(* Logix 5000 project; controller TBIL_All_AOIs_V0_3 vendor 1 type 14 code 176 rev 32.11; software revision 32.00 *)

TASK MainTask (continuous, watchdog 500 ms) : MainProgram
TASK SafetyTask (periodic, rate 20 ms, priority 10, watchdog 20 ms, safety) : SafetyProgram

MODULES
   Local : vendor 1 type 14 code 176 (Compact 0, rev 32.11)
END_MODULES

TYPE Generic_16_Words :
STRUCT
   Data : INT[16];
END_STRUCT
END_TYPE

TYPE Turck_IOLink_Common_Data :
STRUCT
   Read : BOOL;   // For internal use to integrate IOLRead and IOWrite with IOLService
   Write : BOOL;   // For internal use to integrate IOLRead and IOWrite with IOLService
   Reset : BOOL;   // For internal use to integrate IOLRead and IOWrite with IOLService
   Done : BOOL;   // For internal use to integrate IOLRead and IOWrite with IOLService
   Error : BOOL;   // For internal use to integrate IOLRead and IOWrite with IOLService
   Port_in_Use : SINT;   // Each bit is set to show that a port is in use. If it's not in use the port diagnostics will be disabled so IO-Link can still be used but won't throw a red light if no device plugged
   Port : INT;   // For internal use to integrate IOLRead and IOWrite with IOLService
   Index : INT;   // For internal use to integrate IOLRead and IOWrite with IOLService
   SubIndex : INT;   // For internal use to integrate IOLRead and IOWrite with IOLService
   Length : INT;   // For internal use to integrate IOLRead and IOWrite with IOLService
   TicketNum : INT;   // For internal use to integrate IOLRead and IOWrite with IOLService
   Status : INT;   // For internal use to integrate IOLRead and IOWrite with IOLService
   NextTicketNum : INT;   // For internal use to integrate IOLRead and IOWrite with IOLService
   ReceiveData : SINT[255];   // For internal use to integrate IOLRead and IOWrite with IOLService
   SendData : SINT[145];   // For internal use to integrate IOLRead and IOWrite with IOLService
   Vendor_IDs : INT[8];
   Device_IDs : DINT[8];
   WriteData : DINT;
   Process_Input_Data : Generic_16_Words[8];
   Process_Output_Data : Generic_16_Words[8];
END_STRUCT
END_TYPE

ADD_ON_INSTRUCTION IO_Link_Universal_Discrete_Hub   (* revision 1.0 *)
VAR_INPUT
   Port : INT; {required}
END_VAR
VAR_IN_OUT
   Common_Data : Turck_IOLink_Common_Data; {required}
END_VAR
VAR_INPUT
   C0_00_or_7A_Out : BOOL; {visible}
   C0_01_or_7B_Out : BOOL; {visible}
   C1_02_or_5A_Out : BOOL; {visible}
   C1_03_or_5B_Out : BOOL; {visible}
   C2_04_or_3A_Out : BOOL; {visible}
   C2_05_or_3B_Out : BOOL; {visible}
   C3_06_or_1A_Out : BOOL; {visible}
   C3_07_or_1B_Out : BOOL; {visible}
   C4_08_or_8A_Out : BOOL; {visible}
   C4_09_or_8B_Out : BOOL; {visible}
   C5_10_or_6A_Out : BOOL; {visible}
   C5_11_or_6B_Out : BOOL; {visible}
   C6_12_or_4A_Out : BOOL; {visible}
   C6_13_or_4B_Out : BOOL; {visible}
   C7_14_or_2A_Out : BOOL; {visible}
   C7_15_or_2B_Out : BOOL; {visible}
END_VAR
VAR_OUTPUT
   C0_00_or_7A_In : BOOL; {visible}
   C0_01_or_7B_In : BOOL; {visible}
   C1_02_or_5A_In : BOOL; {visible}
   C1_03_or_5B_In : BOOL; {visible}
   C2_04_or_3A_In : BOOL; {visible}
   C2_05_or_3B_In : BOOL; {visible}
   C3_06_or_1A_In : BOOL; {visible}
   C3_07_or_1B_In : BOOL; {visible}
   C4_08_or_8A_In : BOOL; {visible}
   C4_09_or_8B_In : BOOL; {visible}
   C5_10_or_6A_In : BOOL; {visible}
   C5_11_or_6B_In : BOOL; {visible}
   C6_12_or_4A_In : BOOL; {visible}
   C6_13_or_4B_In : BOOL; {visible}
   C7_14_or_2A_In : BOOL; {visible}
   C7_15_or_2B_In : BOOL; {visible}
   TBIL_M1_16DIP : BOOL; {access Read Only}
   TBIL_M1_16DXP : BOOL; {access Read Only}
   TBIL_M1_8DOP : BOOL; {access Read Only}
   TBIL_M1_16DXP_B : BOOL; {access Read Only}
   TBIL_L4_16DXP_AUX : BOOL; {access Read Only}
   TBIL_L5_16DXP_AUX : BOOL;
   TBIL_LL_16DXP_AUX : BOOL; {access Read Only}
   TBIL_S3_8DIP : BOOL; {access Read Only}
   TBIL_S3_8DXP : BOOL; {access Read Only}
   TBIL_S4_8DIP : BOOL; {access Read Only}
   TBIL_S4_8DXP : BOOL; {access Read Only}
   Known_Device_Connected : BOOL; {access Read Only, visible}
   Unknown_Device_or_Missing : BOOL; {access Read Only, visible}
END_VAR
VAR
   Port_Less_One : INT; {access None}
   One : SINT; {access None}
   Port_Bit : SINT; {access None}
   Two : DINT; {access None}
END_VAR

ROUTINE Logic   (* ladder *)
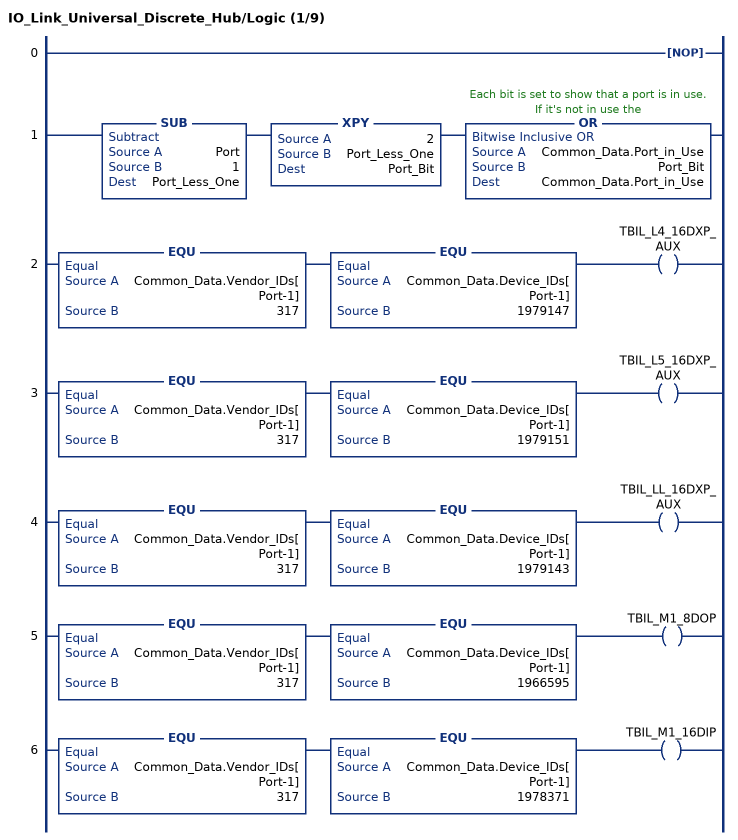
   0: NOP();
   1: SUB(Port,1,Port_Less_One)XPY(2,Port_Less_One,Port_Bit)OR(Common_Data.Port_in_Use,Port_Bit,Common_Data.Port_in_Use);
   2: EQU(Common_Data.Vendor_IDs[Port-1],317)EQU(Common_Data.Device_IDs[Port-1],1979147)OTE(TBIL_L4_16DXP_AUX);
   3: EQU(Common_Data.Vendor_IDs[Port-1],317)EQU(Common_Data.Device_IDs[Port-1],1979151)OTE(TBIL_L5_16DXP_AUX);
   4: EQU(Common_Data.Vendor_IDs[Port-1],317)EQU(Common_Data.Device_IDs[Port-1],1979143)OTE(TBIL_LL_16DXP_AUX);
   5: EQU(Common_Data.Vendor_IDs[Port-1],317)EQU(Common_Data.Device_IDs[Port-1],1966595)OTE(TBIL_M1_8DOP);
   6: EQU(Common_Data.Vendor_IDs[Port-1],317)EQU(Common_Data.Device_IDs[Port-1],1978371)OTE(TBIL_M1_16DIP);
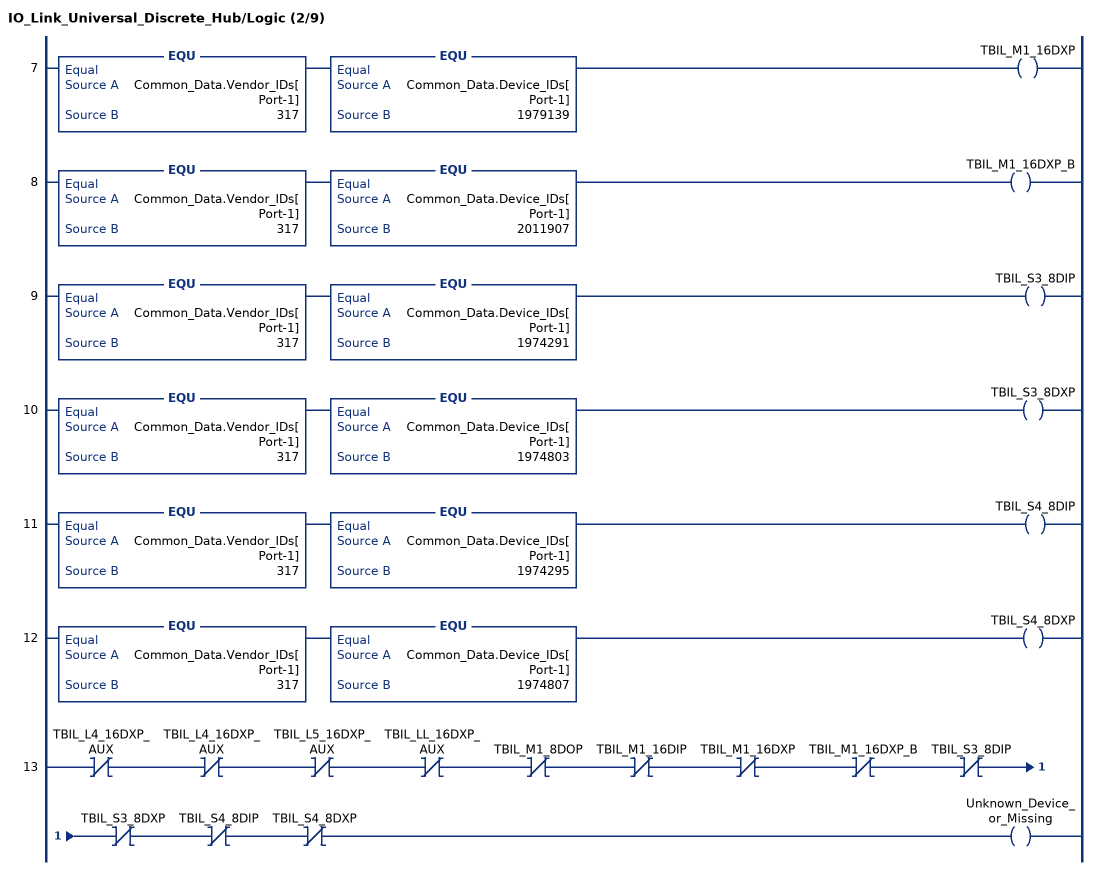
   7: EQU(Common_Data.Vendor_IDs[Port-1],317)EQU(Common_Data.Device_IDs[Port-1],1979139)OTE(TBIL_M1_16DXP);
   8: EQU(Common_Data.Vendor_IDs[Port-1],317)EQU(Common_Data.Device_IDs[Port-1],2011907)OTE(TBIL_M1_16DXP_B);
   9: EQU(Common_Data.Vendor_IDs[Port-1],317)EQU(Common_Data.Device_IDs[Port-1],1974291)OTE(TBIL_S3_8DIP);
   10: EQU(Common_Data.Vendor_IDs[Port-1],317)EQU(Common_Data.Device_IDs[Port-1],1974803)OTE(TBIL_S3_8DXP);
   11: EQU(Common_Data.Vendor_IDs[Port-1],317)EQU(Common_Data.Device_IDs[Port-1],1974295)OTE(TBIL_S4_8DIP);
   12: EQU(Common_Data.Vendor_IDs[Port-1],317)EQU(Common_Data.Device_IDs[Port-1],1974807)OTE(TBIL_S4_8DXP);
   13: XIO(TBIL_L4_16DXP_AUX)XIO(TBIL_L4_16DXP_AUX)XIO(TBIL_L5_16DXP_AUX)XIO(TBIL_LL_16DXP_AUX)XIO(TBIL_M1_8DOP)XIO(TBIL_M1_16DIP)XIO(TBIL_M1_16DXP)XIO(TBIL_M1_16DXP_B)XIO(TBIL_S3_8DIP)XIO(TBIL_S3_8DXP)XIO(TBIL_S4_8DIP)XIO(TBIL_S4_8DXP)OTE(Unknown_Device_or_Missing);
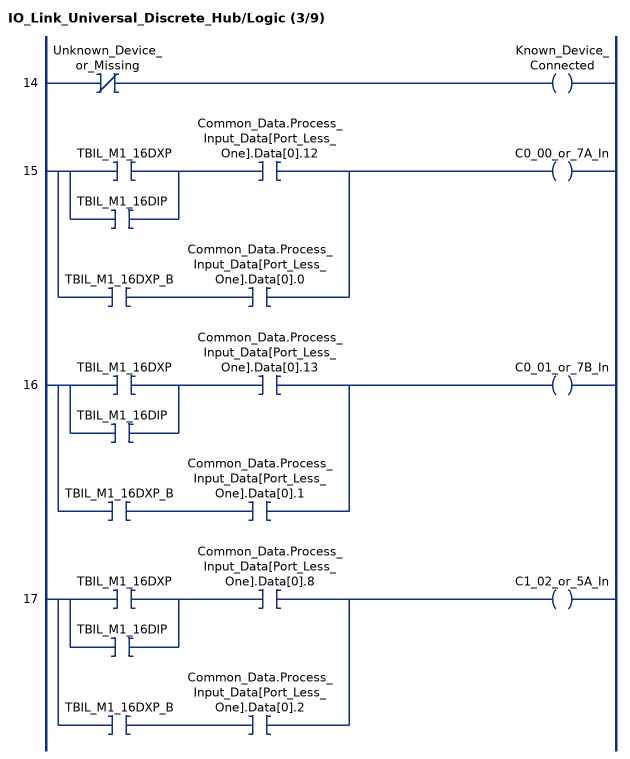
   14: XIO(Unknown_Device_or_Missing)OTE(Known_Device_Connected);
   15: [[XIC(TBIL_M1_16DXP) ,XIC(TBIL_M1_16DIP) ] XIC(Common_Data.Process_Input_Data[Port_Less_One].Data[0].12) ,XIC(TBIL_M1_16DXP_B) XIC(Common_Data.Process_Input_Data[Port_Less_One].Data[0].0) ]OTE(C0_00_or_7A_In);
   16: [[XIC(TBIL_M1_16DXP) ,XIC(TBIL_M1_16DIP) ] XIC(Common_Data.Process_Input_Data[Port_Less_One].Data[0].13) ,XIC(TBIL_M1_16DXP_B) XIC(Common_Data.Process_Input_Data[Port_Less_One].Data[0].1) ]OTE(C0_01_or_7B_In);
   17: [[XIC(TBIL_M1_16DXP) ,XIC(TBIL_M1_16DIP) ] XIC(Common_Data.Process_Input_Data[Port_Less_One].Data[0].8) ,XIC(TBIL_M1_16DXP_B) XIC(Common_Data.Process_Input_Data[Port_Less_One].Data[0].2) ]OTE(C1_02_or_5A_In);
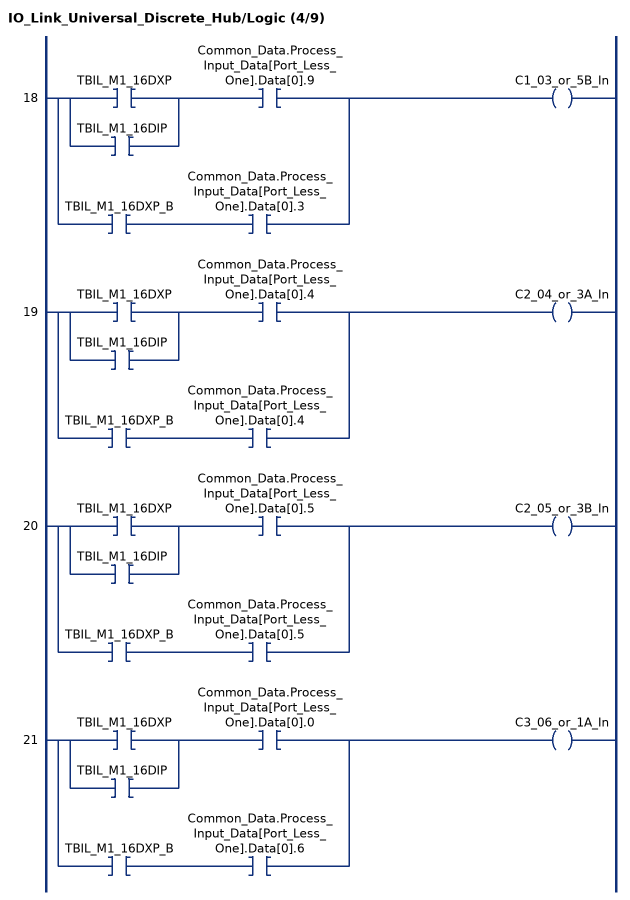
   18: [[XIC(TBIL_M1_16DXP) ,XIC(TBIL_M1_16DIP) ] XIC(Common_Data.Process_Input_Data[Port_Less_One].Data[0].9) ,XIC(TBIL_M1_16DXP_B) XIC(Common_Data.Process_Input_Data[Port_Less_One].Data[0].3) ]OTE(C1_03_or_5B_In);
   19: [[XIC(TBIL_M1_16DXP) ,XIC(TBIL_M1_16DIP) ] XIC(Common_Data.Process_Input_Data[Port_Less_One].Data[0].4) ,XIC(TBIL_M1_16DXP_B) XIC(Common_Data.Process_Input_Data[Port_Less_One].Data[0].4) ]OTE(C2_04_or_3A_In);
   20: [[XIC(TBIL_M1_16DXP) ,XIC(TBIL_M1_16DIP) ] XIC(Common_Data.Process_Input_Data[Port_Less_One].Data[0].5) ,XIC(TBIL_M1_16DXP_B) XIC(Common_Data.Process_Input_Data[Port_Less_One].Data[0].5) ]OTE(C2_05_or_3B_In);
   21: [[XIC(TBIL_M1_16DXP) ,XIC(TBIL_M1_16DIP) ] XIC(Common_Data.Process_Input_Data[Port_Less_One].Data[0].0) ,XIC(TBIL_M1_16DXP_B) XIC(Common_Data.Process_Input_Data[Port_Less_One].Data[0].6) ]OTE(C3_06_or_1A_In);
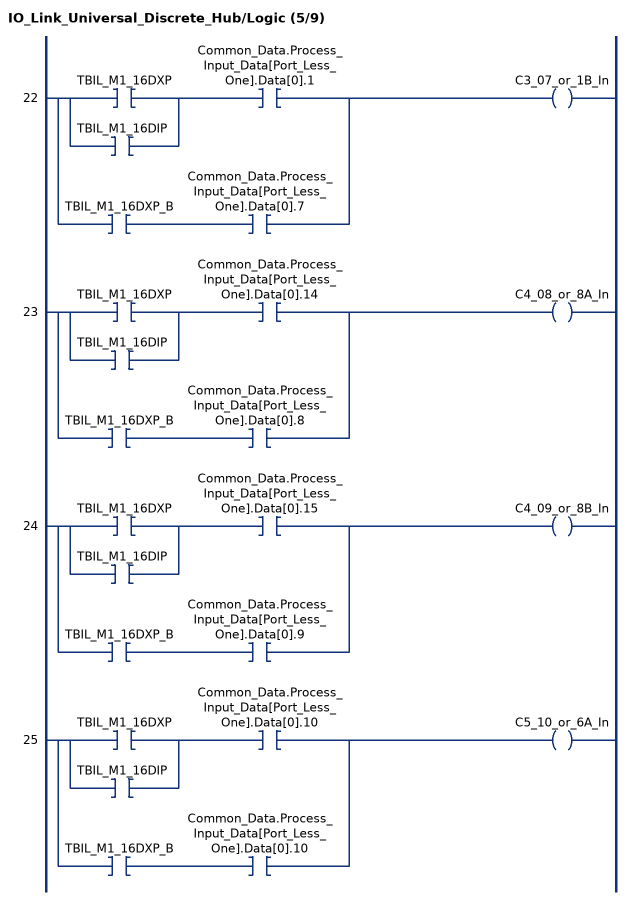
   22: [[XIC(TBIL_M1_16DXP) ,XIC(TBIL_M1_16DIP) ] XIC(Common_Data.Process_Input_Data[Port_Less_One].Data[0].1) ,XIC(TBIL_M1_16DXP_B) XIC(Common_Data.Process_Input_Data[Port_Less_One].Data[0].7) ]OTE(C3_07_or_1B_In);
   23: [[XIC(TBIL_M1_16DXP) ,XIC(TBIL_M1_16DIP) ] XIC(Common_Data.Process_Input_Data[Port_Less_One].Data[0].14) ,XIC(TBIL_M1_16DXP_B) XIC(Common_Data.Process_Input_Data[Port_Less_One].Data[0].8) ]OTE(C4_08_or_8A_In);
   24: [[XIC(TBIL_M1_16DXP) ,XIC(TBIL_M1_16DIP) ] XIC(Common_Data.Process_Input_Data[Port_Less_One].Data[0].15) ,XIC(TBIL_M1_16DXP_B) XIC(Common_Data.Process_Input_Data[Port_Less_One].Data[0].9) ]OTE(C4_09_or_8B_In);
   25: [[XIC(TBIL_M1_16DXP) ,XIC(TBIL_M1_16DIP) ] XIC(Common_Data.Process_Input_Data[Port_Less_One].Data[0].10) ,XIC(TBIL_M1_16DXP_B) XIC(Common_Data.Process_Input_Data[Port_Less_One].Data[0].10) ]OTE(C5_10_or_6A_In);
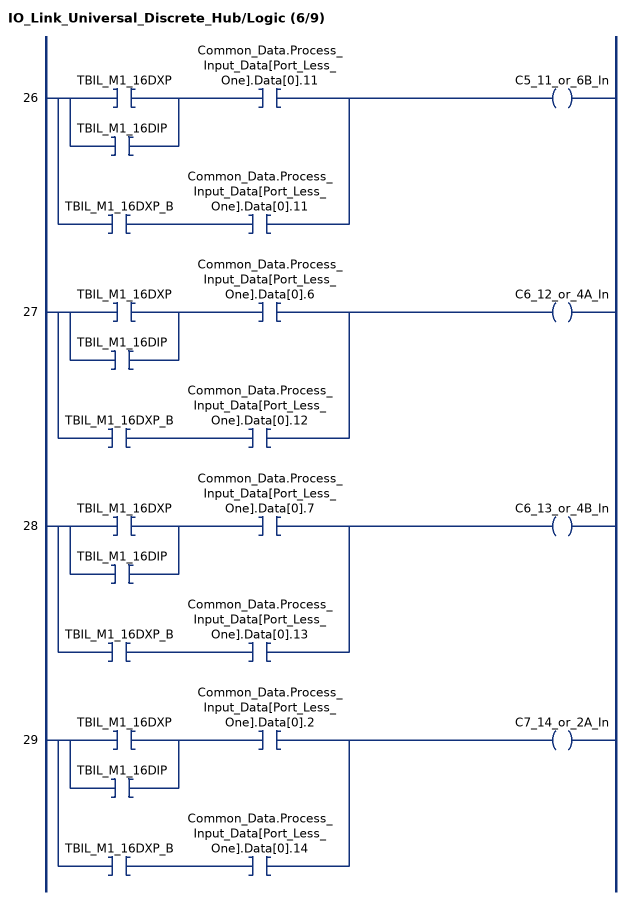
   26: [[XIC(TBIL_M1_16DXP) ,XIC(TBIL_M1_16DIP) ] XIC(Common_Data.Process_Input_Data[Port_Less_One].Data[0].11) ,XIC(TBIL_M1_16DXP_B) XIC(Common_Data.Process_Input_Data[Port_Less_One].Data[0].11) ]OTE(C5_11_or_6B_In);
   27: [[XIC(TBIL_M1_16DXP) ,XIC(TBIL_M1_16DIP) ] XIC(Common_Data.Process_Input_Data[Port_Less_One].Data[0].6) ,XIC(TBIL_M1_16DXP_B) XIC(Common_Data.Process_Input_Data[Port_Less_One].Data[0].12) ]OTE(C6_12_or_4A_In);
   28: [[XIC(TBIL_M1_16DXP) ,XIC(TBIL_M1_16DIP) ] XIC(Common_Data.Process_Input_Data[Port_Less_One].Data[0].7) ,XIC(TBIL_M1_16DXP_B) XIC(Common_Data.Process_Input_Data[Port_Less_One].Data[0].13) ]OTE(C6_13_or_4B_In);
   29: [[XIC(TBIL_M1_16DXP) ,XIC(TBIL_M1_16DIP) ] XIC(Common_Data.Process_Input_Data[Port_Less_One].Data[0].2) ,XIC(TBIL_M1_16DXP_B) XIC(Common_Data.Process_Input_Data[Port_Less_One].Data[0].14) ]OTE(C7_14_or_2A_In);
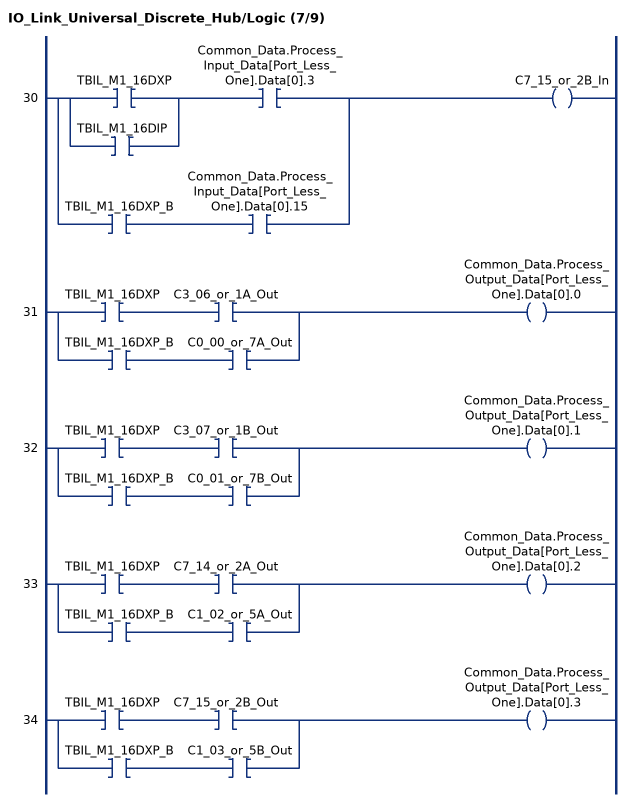
   30: [[XIC(TBIL_M1_16DXP) ,XIC(TBIL_M1_16DIP) ] XIC(Common_Data.Process_Input_Data[Port_Less_One].Data[0].3) ,XIC(TBIL_M1_16DXP_B) XIC(Common_Data.Process_Input_Data[Port_Less_One].Data[0].15) ]OTE(C7_15_or_2B_In);
   31: [XIC(TBIL_M1_16DXP) XIC(C3_06_or_1A_Out) ,XIC(TBIL_M1_16DXP_B) XIC(C0_00_or_7A_Out) ]OTE(Common_Data.Process_Output_Data[Port_Less_One].Data[0].0);
   32: [XIC(TBIL_M1_16DXP) XIC(C3_07_or_1B_Out) ,XIC(TBIL_M1_16DXP_B) XIC(C0_01_or_7B_Out) ]OTE(Common_Data.Process_Output_Data[Port_Less_One].Data[0].1);
   33: [XIC(TBIL_M1_16DXP) XIC(C7_14_or_2A_Out) ,XIC(TBIL_M1_16DXP_B) XIC(C1_02_or_5A_Out) ]OTE(Common_Data.Process_Output_Data[Port_Less_One].Data[0].2);
   34: [XIC(TBIL_M1_16DXP) XIC(C7_15_or_2B_Out) ,XIC(TBIL_M1_16DXP_B) XIC(C1_03_or_5B_Out) ]OTE(Common_Data.Process_Output_Data[Port_Less_One].Data[0].3);
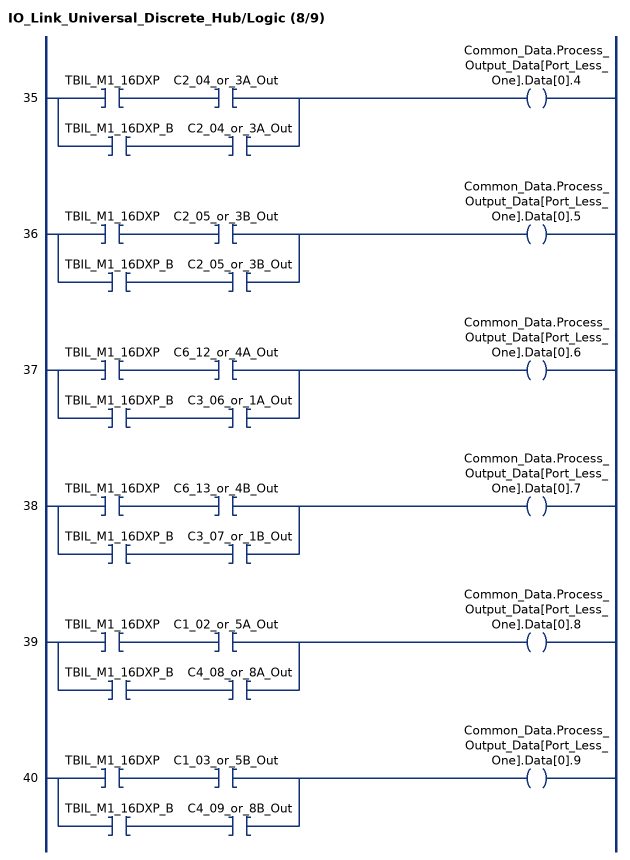
   35: [XIC(TBIL_M1_16DXP) XIC(C2_04_or_3A_Out) ,XIC(TBIL_M1_16DXP_B) XIC(C2_04_or_3A_Out) ]OTE(Common_Data.Process_Output_Data[Port_Less_One].Data[0].4);
   36: [XIC(TBIL_M1_16DXP) XIC(C2_05_or_3B_Out) ,XIC(TBIL_M1_16DXP_B) XIC(C2_05_or_3B_Out) ]OTE(Common_Data.Process_Output_Data[Port_Less_One].Data[0].5);
   37: [XIC(TBIL_M1_16DXP) XIC(C6_12_or_4A_Out) ,XIC(TBIL_M1_16DXP_B) XIC(C3_06_or_1A_Out) ]OTE(Common_Data.Process_Output_Data[Port_Less_One].Data[0].6);
   38: [XIC(TBIL_M1_16DXP) XIC(C6_13_or_4B_Out) ,XIC(TBIL_M1_16DXP_B) XIC(C3_07_or_1B_Out) ]OTE(Common_Data.Process_Output_Data[Port_Less_One].Data[0].7);
   39: [XIC(TBIL_M1_16DXP) XIC(C1_02_or_5A_Out) ,XIC(TBIL_M1_16DXP_B) XIC(C4_08_or_8A_Out) ]OTE(Common_Data.Process_Output_Data[Port_Less_One].Data[0].8);
   40: [XIC(TBIL_M1_16DXP) XIC(C1_03_or_5B_Out) ,XIC(TBIL_M1_16DXP_B) XIC(C4_09_or_8B_Out) ]OTE(Common_Data.Process_Output_Data[Port_Less_One].Data[0].9);
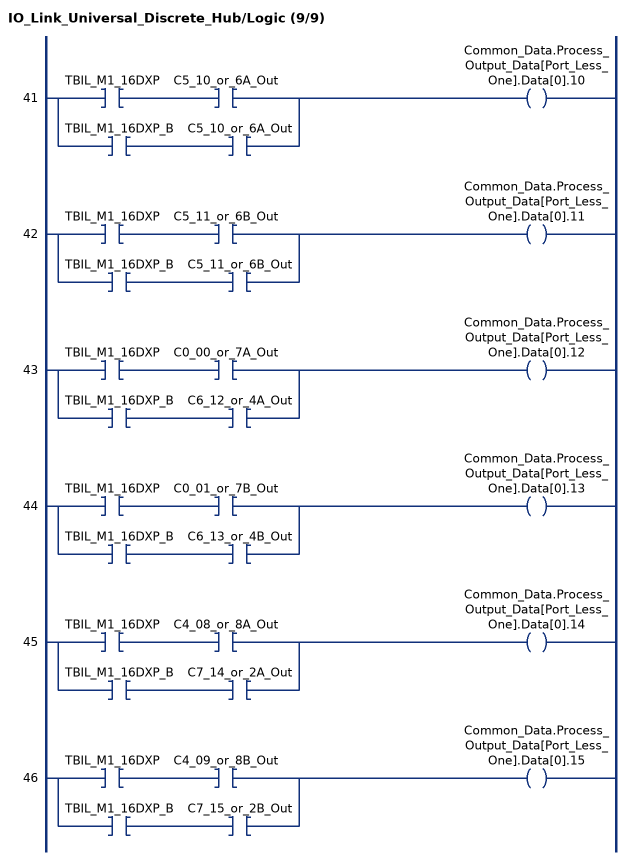
   41: [XIC(TBIL_M1_16DXP) XIC(C5_10_or_6A_Out) ,XIC(TBIL_M1_16DXP_B) XIC(C5_10_or_6A_Out) ]OTE(Common_Data.Process_Output_Data[Port_Less_One].Data[0].10);
   42: [XIC(TBIL_M1_16DXP) XIC(C5_11_or_6B_Out) ,XIC(TBIL_M1_16DXP_B) XIC(C5_11_or_6B_Out) ]OTE(Common_Data.Process_Output_Data[Port_Less_One].Data[0].11);
   43: [XIC(TBIL_M1_16DXP) XIC(C0_00_or_7A_Out) ,XIC(TBIL_M1_16DXP_B) XIC(C6_12_or_4A_Out) ]OTE(Common_Data.Process_Output_Data[Port_Less_One].Data[0].12);
   44: [XIC(TBIL_M1_16DXP) XIC(C0_01_or_7B_Out) ,XIC(TBIL_M1_16DXP_B) XIC(C6_13_or_4B_Out) ]OTE(Common_Data.Process_Output_Data[Port_Less_One].Data[0].13);
   45: [XIC(TBIL_M1_16DXP) XIC(C4_08_or_8A_Out) ,XIC(TBIL_M1_16DXP_B) XIC(C7_14_or_2A_Out) ]OTE(Common_Data.Process_Output_Data[Port_Less_One].Data[0].14);
   46: [XIC(TBIL_M1_16DXP) XIC(C4_09_or_8B_Out) ,XIC(TBIL_M1_16DXP_B) XIC(C7_15_or_2B_Out) ]OTE(Common_Data.Process_Output_Data[Port_Less_One].Data[0].15);
END_ROUTINE
END_ADD_ON_INSTRUCTION

ADD_ON_INSTRUCTION TBEN_Lx_8IOL_AOI   (* revision 0.1 Unreleased, ExecutePrescan *)
// Create an AOI specific to TBEN-Lx-8IOL devices
// Revision note:
// V0_1 Initial Approach
// V0_2 Cleaning Up
// Help:
// IOL_Service - used with Turck BL20, BL67, BLC and TBEN IOLink masters to process requests from IOL_ReadString, IOL_WriteString, IOL_ReadData and IOL_WriteData AOI's.
// Status	Description
// 0	Operation completed successfully
// 	Status = 100 - 102, Ethernet IP MSG instruction errors - check communication parameters
// 100	IOL_SendMSG completed with error, check communication parameters
// 101	IOL_RecevieMSG completed with error, check communication parameters
// 110	IOL_Service Retry Limit exceeded
// 111	Slot specified not an IOLink master
// 	Status = 1000 to 1255, no response from device, connection error
// 1016	Device not connected or Port not configured as IOLink port
// 	Status = 2000 to 2255,  device response indicates error
// 2000	Device error, no details
// 2017	Device error, Index not available
// 2018	Device error, Subindex not available
// 2032	Device error, Service temporarily not available
// 2033	Device error, Service temporarily not available - local control
// 2034	Device error, Service temporarily not available - device control
// 2035	Device error, Index not writeable
// 2048	Device error, Parameter value out of range
// 2049	Device error, Parameter value above limit
// 2050	Device error, Parameter value below limit
// 2051	Device error, Parameter value length overrun (check IOLWrite precision/string length)
// 2052	Device error, Parameter value length underrun (check IOLWrite precision/string length)
// 2053	Device error, Function not available
// 2054	Device error, Function temporarily not available
// 2064	Device error, Parameter set invalid
// 2065	Device error, Inconsistent parameter set
// 2130	Device error, Application not ready
// 	Status = 3000 to 3255,   device response indicates vendor specific error
// 3000	Vendor specific error, no details
// 3001	Vendor specific error, vendor specific error number
// 3255	Vendor specific error, vendor specific error number
// 	Status = 7000 to 7255,  IOL-M Error Codes
// 7000	Unexpected write request instead of read request
// 7001	Decode error
// 7002	Port occupied by another task
// 	Status = 8000 to 8255,  IOL-M Error Codes
// 8000	Timeout when IOL-Ds or IOL-M ports are busy
// 8001	IOL Index out of range
// 8002	Port address greater than maximum
// 8003	Port function not supported
VAR_IN_OUT
   Common_Data : Turck_IOLink_Common_Data; {required}
        .SendData[1]   // For internal use to integrate IOLRead and IOLWrite with IOLService
   IOL_Read_MSG : MESSAGE; {required}
   IOL_Write_MSG : MESSAGE; {required}
   TBEN_I_DATA : INT[173]; {required}   // Input Data from IO Block
   TBEN_O_DATA : INT[131]; {required}   // Output Data to IO Block
   TBEN_C_DATA : SINT[160]; {required}
END_VAR
VAR_OUTPUT
   DXP1_OUT : BOOL; {visible}
   DXP3_OUT : BOOL; {visible}
   DXP5_OUT : BOOL; {visible}
   DXP7_OUT : BOOL; {visible}
   IOLDevice_PORT1 : BOOL; {visible}
   IOLDevice_PORT2 : BOOL; {visible}
   IOLDevice_PORT3 : BOOL; {visible}
   IOLDevice_PORT4 : BOOL; {visible}
   IOLDevice_PORT5 : BOOL; {visible}
   IOLDevice_PORT6 : BOOL; {visible}
   IOLDevice_PORT7 : BOOL; {visible}
   IOLDevice_PORT8 : BOOL; {visible}
END_VAR
VAR_INPUT
   IOL0_DI : BOOL; {visible}
   DXP1_IN : BOOL; {visible}
   IOL2_DI : BOOL; {visible}
   DXP3_IN : BOOL; {visible}
   IOL4_DI : BOOL; {visible}
   DXP5_IN : BOOL; {visible}
   IOL6_DI : BOOL; {visible}
   DXP7_IN : BOOL; {visible}
   IOL8_DI : BOOL; {visible}
   IOL10_DI : BOOL; {visible}
   IOL12_DI : BOOL; {visible}
   IOL14_DI : BOOL; {visible}
   PORT1_Mode_IOL_or_DI : BOOL;   // 0: IO-LINK without validation 1: Port is set to DI (Power Cycle or Module Inhibit cycle require)
   PORT2_Mode_IOL_or_DI : BOOL;   // 0: IO-LINK without validation 1: Port is set to DI (Power Cycle or Module Inhibit cycle require)
   PORT3_Mode_IOL_or_DI : BOOL;   // 0: IO-LINK without validation 1: Port is set to DI (Power Cycle or Module Inhibit cycle require)
   PORT4_Mode_IOL_or_DI : BOOL;   // 0: IO-LINK without validation 1: Port is set to DI (Power Cycle or Module Inhibit cycle require)
   PORT5_Mode_IOL_or_DI : BOOL;   // 0: IO-LINK without validation 1: Port is set to DI (Power Cycle or Module Inhibit cycle require)
   PORT6_Mode_IOL_or_DI : BOOL;   // 0: IO-LINK without validation 1: Port is set to DI (Power Cycle or Module Inhibit cycle require)
   PORT7_Mode_IOL_or_DI : BOOL;   // 0: IO-LINK without validation 1: Port is set to DI (Power Cycle or Module Inhibit cycle require)
   PORT8_Mode_IOL_or_DI : BOOL;   // 0: IO-LINK without validation 1: Port is set to DI (Power Cycle or Module Inhibit cycle require)
   DisableOutput_DXP1 : BOOL;
   DisableOutput_DXP3 : BOOL;
   DisableOutput_DXP5 : BOOL;
   DisableOutput_DXP7 : BOOL;
END_VAR
VAR_OUTPUT
   Device_Restart_Required : BOOL; {visible}
END_VAR
VAR_INPUT
   DeviceStatus : DINT;
END_VAR
VAR
   IOLReadActive : BOOL;
   IOLWriteActive : BOOL;
   RetryCount : DINT;
   IOL_Error_Count : DINT; {access None}
   IOLReset_ONS : BOOL; {access None}
   ER1 : BOOL; {access None}
   ER2 : BOOL; {access None}
   tempReceiveData : SINT[255]; {access None}
   Generate_Status : BOOL; {access None}
   ABS_RD_0 : INT; {access None}
   ABS_RD_1 : INT; {access None}
   ABS_RD_2 : INT; {access None}
   ABS_RD_3 : INT; {access None}
   tempSendData : SINT[145]; {access None}
   IOL_READ_Request : BOOL; {access None}
   IOL_WRITE_Request : BOOL; {access None}
   StartupDone : BOOL; {access None}
   Done : BOOL; {access None}
   Error : BOOL; {access None}
   Active : BOOL; {access None}
   Pending : BOOL; {access None}
   Pending_or_Active : BOOL; {access None}
   StartupCount : SINT; {access None}
   DoneCount : SINT; {access None}
   MyTicketNum : INT; {access None}
   Update_Data : BOOL; {access None}
   Read_ONS : BOOL; {access None}
   ReadRequest : BOOL; {access None}
   Prev_Input_Data_Valids : INT; {access None}
   Status : DINT; {access None}
   ErrorCount : DINT; {access None}
   PIDV_Delay : TIMER := (PRE := 1000); {access None}
   TimeDelay : TIMER := (PRE := 500); {access None}
END_VAR

ROUTINE Logic   (* ladder *)
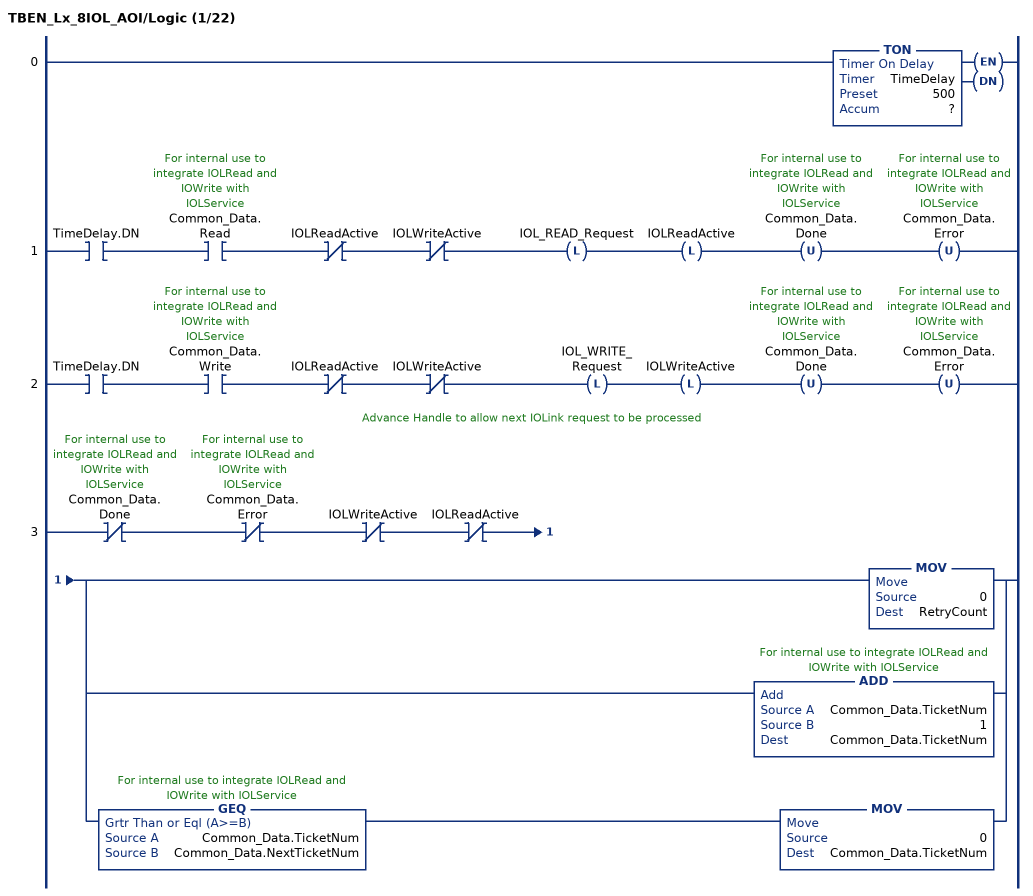
   0: TON(TimeDelay,?,?);
   1: XIC(TimeDelay.DN)XIC(Common_Data.Read)XIO(IOLReadActive)XIO(IOLWriteActive)OTL(IOL_READ_Request)OTL(IOLReadActive)OTU(Common_Data.Done)OTU(Common_Data.Error);
   2: XIC(TimeDelay.DN)XIC(Common_Data.Write)XIO(IOLReadActive)XIO(IOLWriteActive)OTL(IOL_WRITE_Request)OTL(IOLWriteActive)OTU(Common_Data.Done)OTU(Common_Data.Error);
   // Advance Handle to allow next IOLink request to be processed
   3: XIO(Common_Data.Done)XIO(Common_Data.Error)XIO(IOLWriteActive)XIO(IOLReadActive)[MOV(0,RetryCount) ,ADD(Common_Data.TicketNum,1,Common_Data.TicketNum) ,GEQ(Common_Data.TicketNum,Common_Data.NextTicketNum) MOV(0,Common_Data.TicketNum) ];
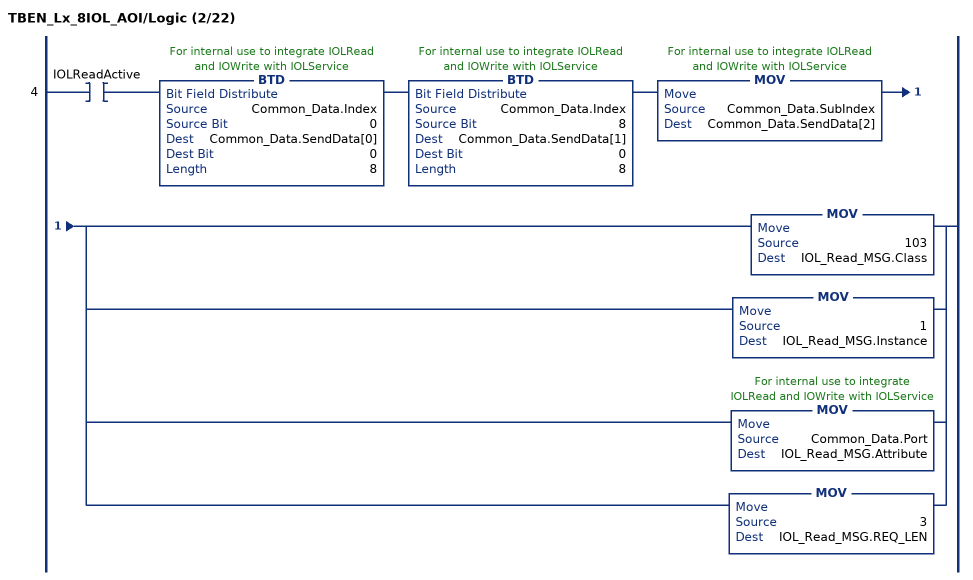
   4: XIC(IOLReadActive)BTD(Common_Data.Index,0,Common_Data.SendData[0],0,8)BTD(Common_Data.Index,8,Common_Data.SendData[1],0,8)MOV(Common_Data.SubIndex,Common_Data.SendData[2])[MOV(103,IOL_Read_MSG.Class) ,MOV(1,IOL_Read_MSG.Instance) ,MOV(Common_Data.Port,IOL_Read_MSG.Attribute) ,MOV(3,IOL_Read_MSG.REQ_LEN) ];
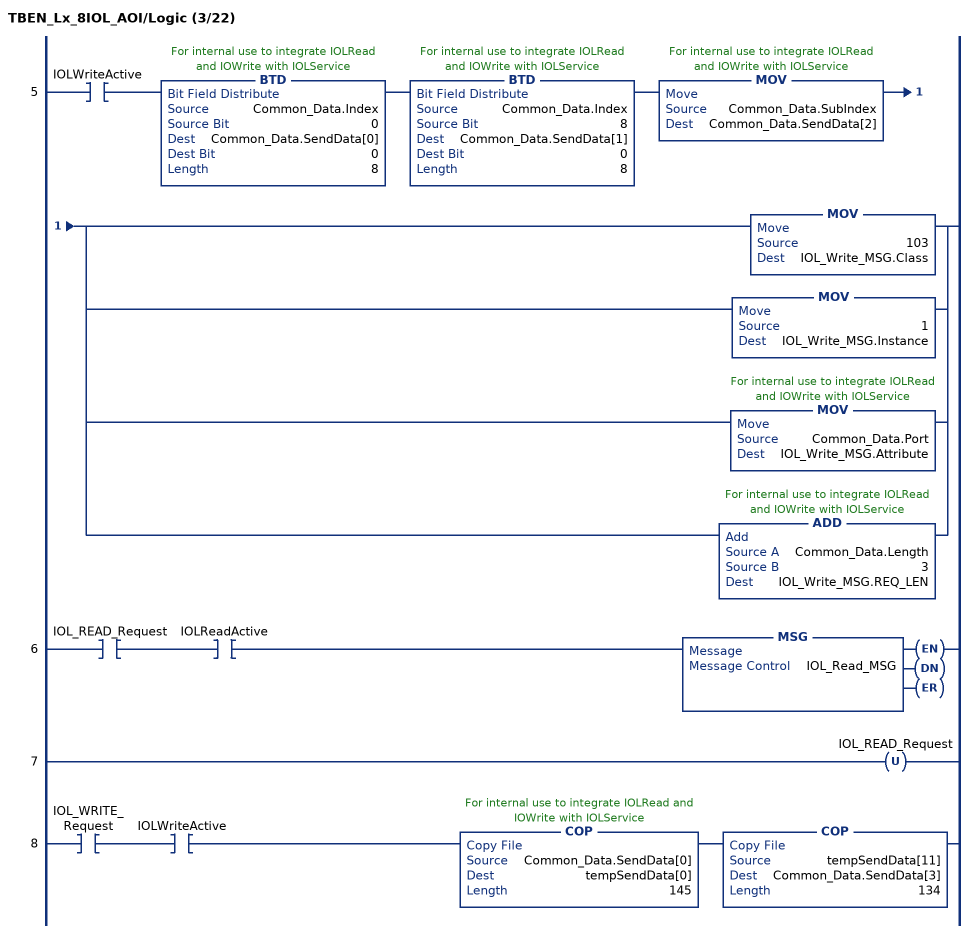
   5: XIC(IOLWriteActive)BTD(Common_Data.Index,0,Common_Data.SendData[0],0,8)BTD(Common_Data.Index,8,Common_Data.SendData[1],0,8)MOV(Common_Data.SubIndex,Common_Data.SendData[2])[MOV(103,IOL_Write_MSG.Class) ,MOV(1,IOL_Write_MSG.Instance) ,MOV(Common_Data.Port,IOL_Write_MSG.Attribute) ,ADD(Common_Data.Length,3,IOL_Write_MSG.REQ_LEN) ];
   6: XIC(IOL_READ_Request)XIC(IOLReadActive)MSG(IOL_Read_MSG);
   7: OTU(IOL_READ_Request);
   8: XIC(IOL_WRITE_Request)XIC(IOLWriteActive)COP(Common_Data.SendData[0],tempSendData[0],145)COP(tempSendData[11],Common_Data.SendData[3],134);
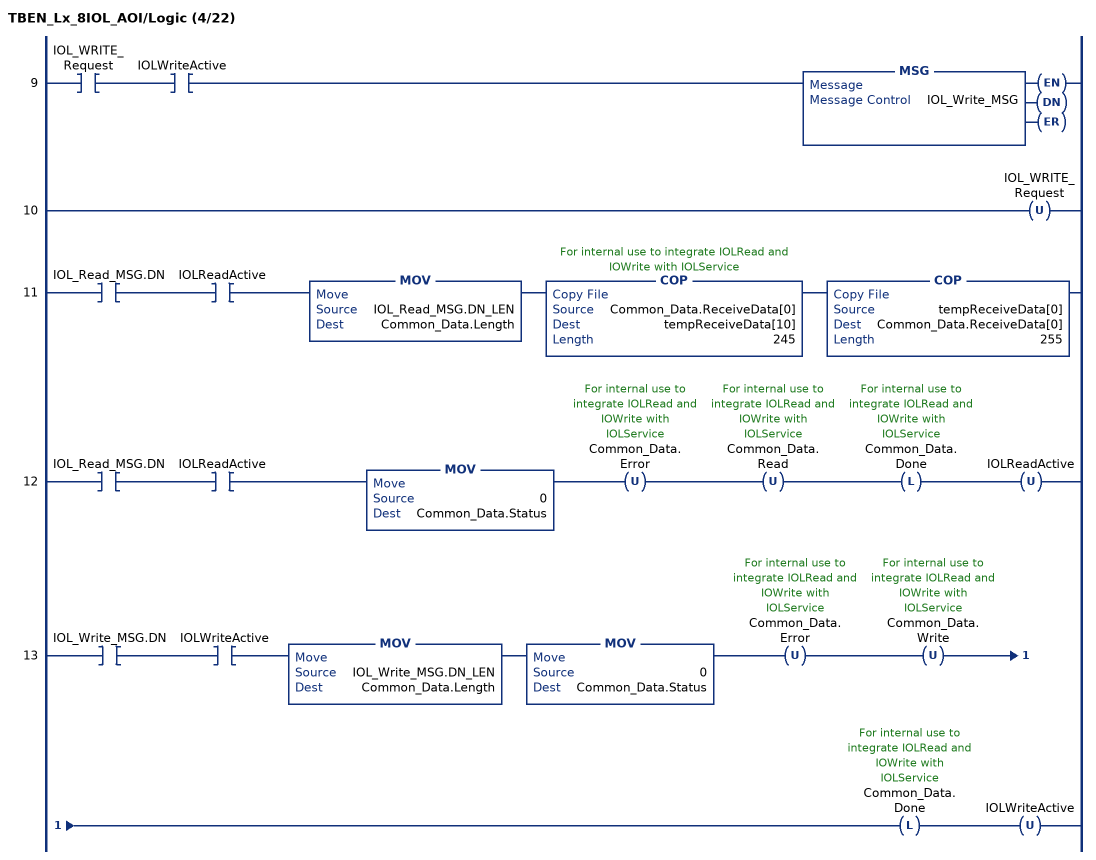
   9: XIC(IOL_WRITE_Request)XIC(IOLWriteActive)MSG(IOL_Write_MSG);
   10: OTU(IOL_WRITE_Request);
   11: XIC(IOL_Read_MSG.DN)XIC(IOLReadActive)MOV(IOL_Read_MSG.DN_LEN,Common_Data.Length)COP(Common_Data.ReceiveData[0],tempReceiveData[10],245)COP(tempReceiveData[0],Common_Data.ReceiveData[0],255);
   12: XIC(IOL_Read_MSG.DN)XIC(IOLReadActive)MOV(0,Common_Data.Status)OTU(Common_Data.Error)OTU(Common_Data.Read)OTL(Common_Data.Done)OTU(IOLReadActive);
   13: XIC(IOL_Write_MSG.DN)XIC(IOLWriteActive)MOV(IOL_Write_MSG.DN_LEN,Common_Data.Length)MOV(0,Common_Data.Status)OTU(Common_Data.Error)OTU(Common_Data.Write)OTL(Common_Data.Done)OTU(IOLWriteActive);
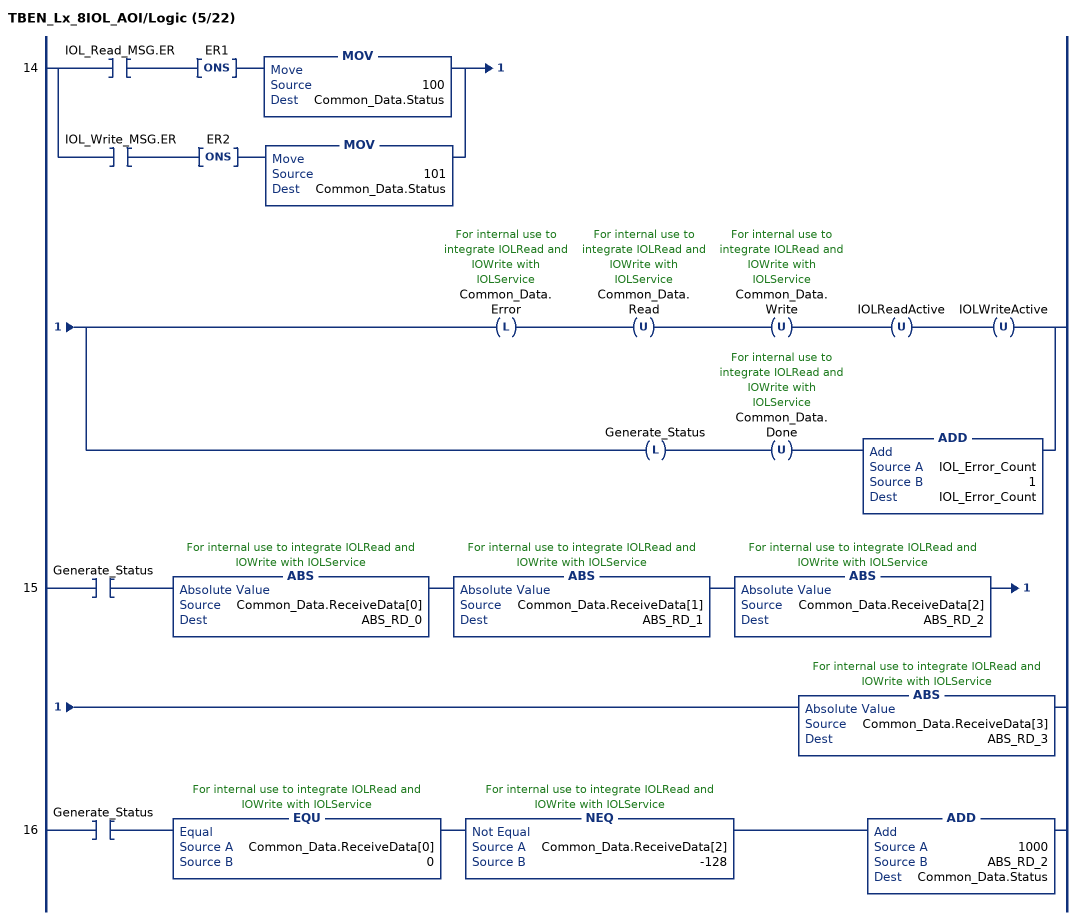
   14: [XIC(IOL_Read_MSG.ER) ONS(ER1) MOV(100,Common_Data.Status) ,XIC(IOL_Write_MSG.ER) ONS(ER2) MOV(101,Common_Data.Status) ][OTL(Common_Data.Error) OTU(Common_Data.Read) OTU(Common_Data.Write) OTU(IOLReadActive) OTU(IOLWriteActive) ,OTL(Generate_Status) OTU(Common_Data.Done) ADD(IOL_Error_Count,1,IOL_Error_Count) ];
   15: XIC(Generate_Status)ABS(Common_Data.ReceiveData[0],ABS_RD_0)ABS(Common_Data.ReceiveData[1],ABS_RD_1)ABS(Common_Data.ReceiveData[2],ABS_RD_2)ABS(Common_Data.ReceiveData[3],ABS_RD_3);
   16: XIC(Generate_Status)EQU(Common_Data.ReceiveData[0],0)NEQ(Common_Data.ReceiveData[2],-128)ADD(1000,ABS_RD_2,Common_Data.Status);
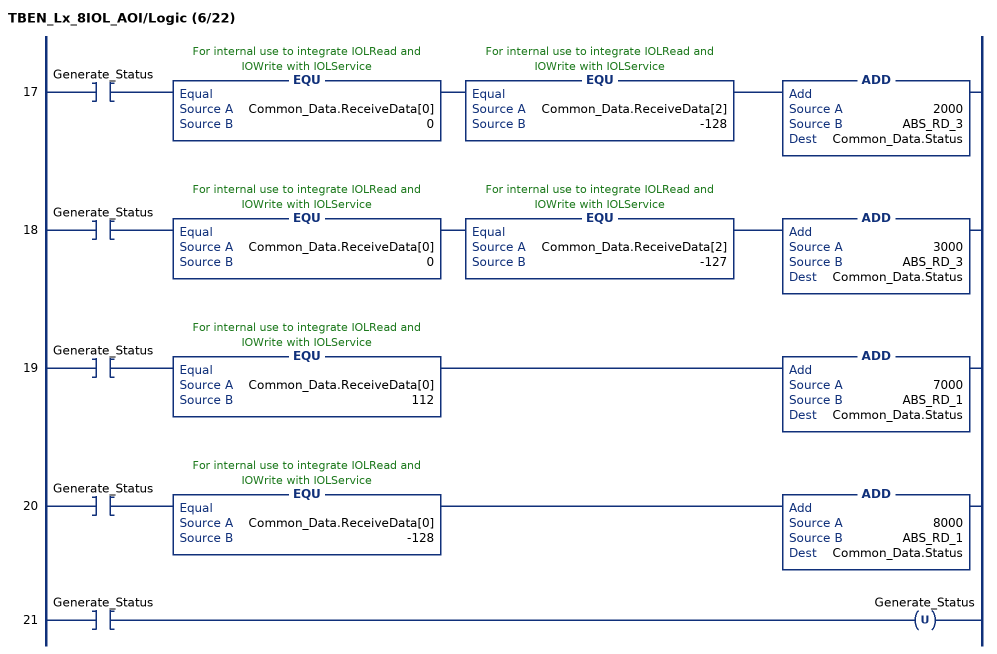
   17: XIC(Generate_Status)EQU(Common_Data.ReceiveData[0],0)EQU(Common_Data.ReceiveData[2],-128)ADD(2000,ABS_RD_3,Common_Data.Status);
   18: XIC(Generate_Status)EQU(Common_Data.ReceiveData[0],0)EQU(Common_Data.ReceiveData[2],-127)ADD(3000,ABS_RD_3,Common_Data.Status);
   19: XIC(Generate_Status)EQU(Common_Data.ReceiveData[0],112)ADD(7000,ABS_RD_1,Common_Data.Status);
   20: XIC(Generate_Status)EQU(Common_Data.ReceiveData[0],-128)ADD(8000,ABS_RD_1,Common_Data.Status);
   21: XIC(Generate_Status)OTU(Generate_Status);
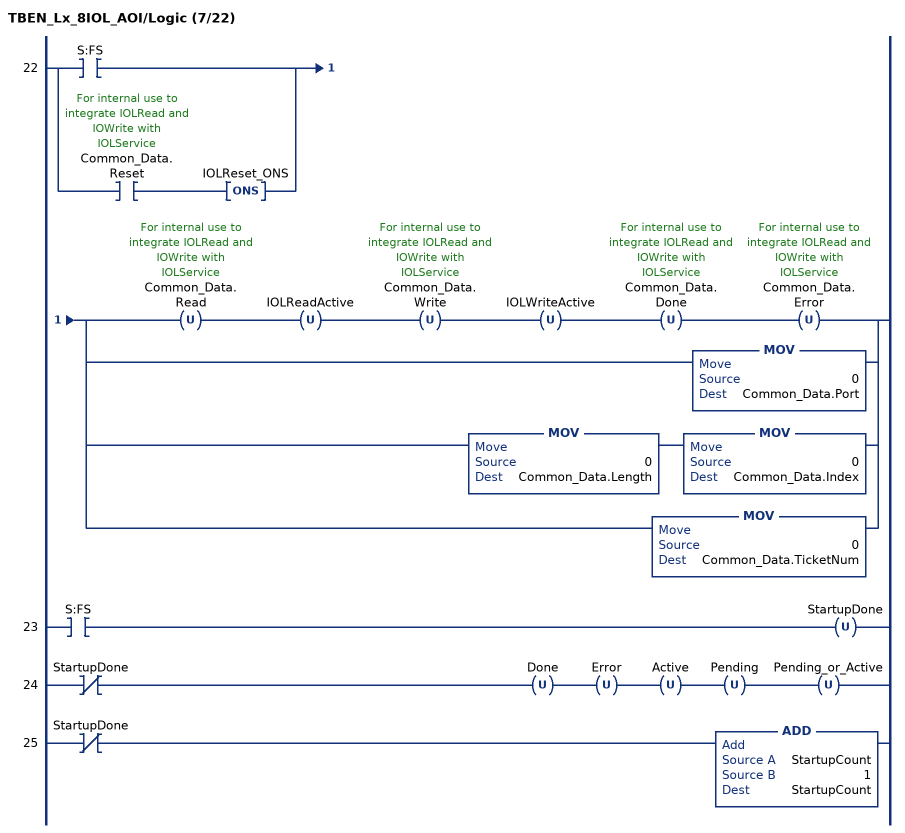
   22: [XIC(S:FS) ,XIC(Common_Data.Reset) ONS(IOLReset_ONS) ][OTU(Common_Data.Read) OTU(IOLReadActive) OTU(Common_Data.Write) OTU(IOLWriteActive) OTU(Common_Data.Done) OTU(Common_Data.Error) ,MOV(0,Common_Data.Port) ,MOV(0,Common_Data.Length) MOV(0,Common_Data.Index) ,MOV(0,Common_Data.TicketNum) ];
   23: XIC(S:FS)OTU(StartupDone);
   24: XIO(StartupDone)OTU(Done)OTU(Error)OTU(Active)OTU(Pending)OTU(Pending_or_Active);
   25: XIO(StartupDone)ADD(StartupCount,1,StartupCount);
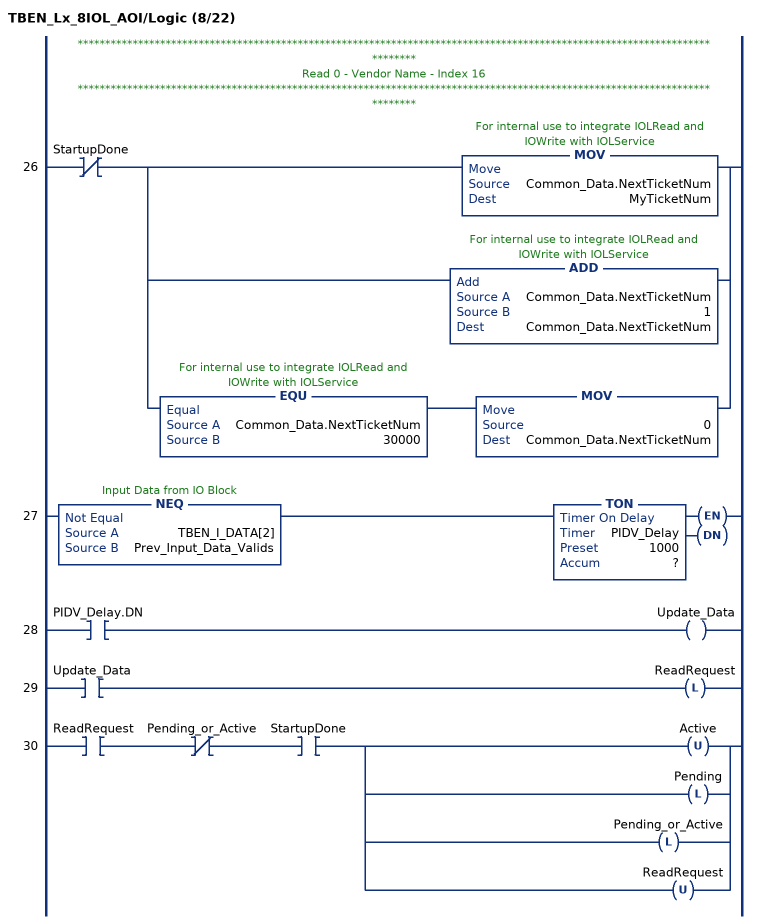
   // ***************************************************************************************************************************
   // Read 0 - Vendor Name - Index 16
   // ***************************************************************************************************************************
   26: XIO(StartupDone)[MOV(Common_Data.NextTicketNum,MyTicketNum) ,ADD(Common_Data.NextTicketNum,1,Common_Data.NextTicketNum) ,EQU(Common_Data.NextTicketNum,30000) MOV(0,Common_Data.NextTicketNum) ];
   27: NEQ(TBEN_I_DATA[2],Prev_Input_Data_Valids)TON(PIDV_Delay,?,?);
   28: XIC(PIDV_Delay.DN)OTE(Update_Data);
   29: XIC(Update_Data)OTL(ReadRequest);
   30: XIC(ReadRequest)XIO(Pending_or_Active)XIC(StartupDone)[OTU(Active) ,OTL(Pending) ,OTL(Pending_or_Active) ,OTU(ReadRequest) ];
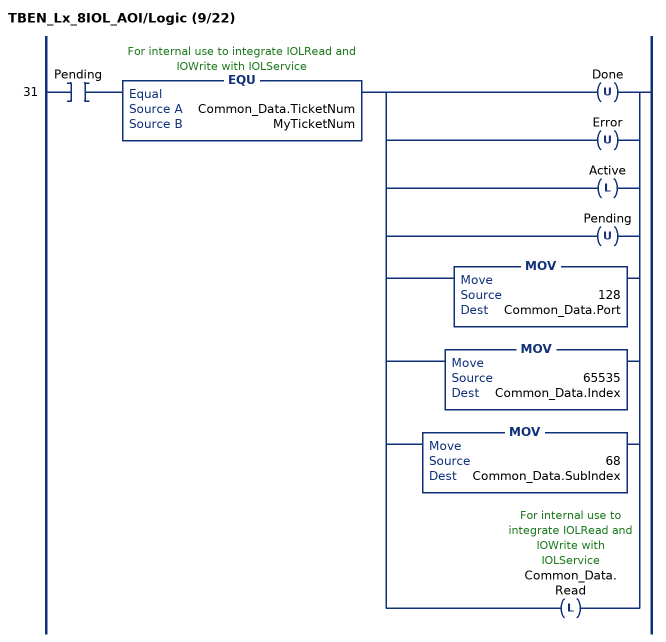
   31: XIC(Pending)EQU(Common_Data.TicketNum,MyTicketNum)[OTU(Done) ,OTU(Error) ,OTL(Active) ,OTU(Pending) ,MOV(128,Common_Data.Port) ,MOV(65535,Common_Data.Index) ,MOV(68,Common_Data.SubIndex) ,OTL(Common_Data.Read) ];
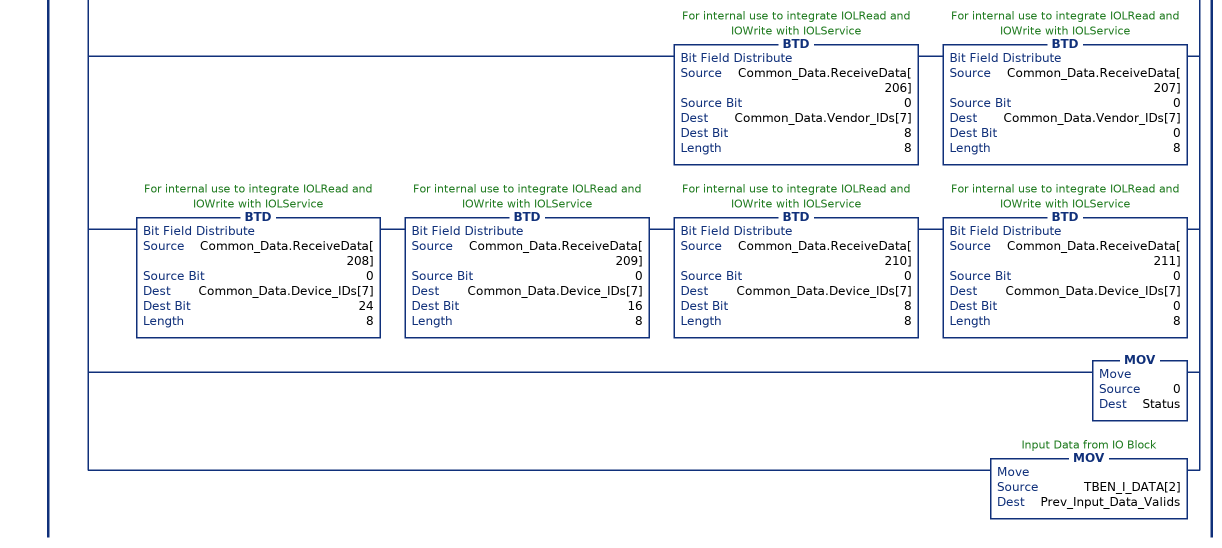
   32: XIC(Active)XIC(Common_Data.Done)[OTL(Done) ,ADD(DoneCount,1,DoneCount) ,OTU(Error) ,OTU(Active) ,OTU(Pending) ,OTU(Pending_or_Active) ,OTU(Common_Data.Done) ,BTD(Common_Data.ReceiveData[10],0,Common_Data.Vendor_IDs[0],8,8) BTD(Common_Data.ReceiveData[11],0,Common_Data.Vendor_IDs[0],0,8) ,BTD(Common_Data.ReceiveData[12],0,Common_Data.Device_IDs[0],24,8) BTD(Common_Data.ReceiveData[13],0,Common_Data.Device_IDs[0],16,8) BTD(Common_Data.ReceiveData[14],0,Common_Data.Device_IDs[0],8,8) BTD(Common_Data.ReceiveData[15],0,Common_Data.Device_IDs[0],0,8) ,BTD(Common_Data.ReceiveData[38],0,Common_Data.Vendor_IDs[1],8,8) BTD(Common_Data.ReceiveData[39],0,Common_Data.Vendor_IDs[1],0,8) ,BTD(Common_Data.ReceiveData[40],0,Common_Data.Device_IDs[1],24,8) BTD(Common_Data.ReceiveData[41],0,Common_Data.Device_IDs[1],16,8) BTD(Common_Data.ReceiveData[42],0,Common_Data.Device_IDs[1],8,8) BTD(Common_Data.ReceiveData[43],0,Common_Data.Device_IDs[1],0,8) ,BTD(Common_Data.ReceiveData[66],0,Common_Data.Vendor_IDs[2],8,8) BTD(Common_Data.ReceiveData[67],0,Common_Data.Vendor_IDs[2],0,8) ,BTD(Common_Data.ReceiveData[68],0,Common_Data.Device_IDs[2],24,8) BTD(Common_Data.ReceiveData[69],0,Common_Data.Device_IDs[2],16,8) BTD(Common_Data.ReceiveData[70],0,Common_Data.Device_IDs[2],8,8) BTD(Common_Data.ReceiveData[71],0,Common_Data.Device_IDs[2],0,8) ,BTD(Common_Data.ReceiveData[94],0,Common_Data.Vendor_IDs[3],8,8) BTD(Common_Data.ReceiveData[95],0,Common_Data.Vendor_IDs[3],0,8) ,BTD(Common_Data.ReceiveData[96],0,Common_Data.Device_IDs[3],24,8) BTD(Common_Data.ReceiveData[97],0,Common_Data.Device_IDs[3],16,8) BTD(Common_Data.ReceiveData[98],0,Common_Data.Device_IDs[3],8,8) BTD(Common_Data.ReceiveData[99],0,Common_Data.Device_IDs[3],0,8) ,BTD(Common_Data.ReceiveData[122],0,Common_Data.Vendor_IDs[4],8,8) BTD(Common_Data.ReceiveData[123],0,Common_Data.Vendor_IDs[4],0,8) ,BTD(Common_Data.ReceiveData[124],0,Common_Data.Device_IDs[4],24,8) BTD(Common_Data.ReceiveData[125],0,Common_Data.Device_IDs[4],16,8) BTD(Common_Data.ReceiveData[126],0,Common_Data.Device_IDs[4],8,8) BTD(Common_Data.ReceiveData[127],0,Common_Data.Device_IDs[4],0,8) ,BTD(Common_Data.ReceiveData[150],0,Common_Data.Vendor_IDs[5],8,8) BTD(Common_Data.ReceiveData[151],0,Common_Data.Vendor_IDs[5],0,8) ,BTD(Common_Data.ReceiveData[152],0,Common_Data.Device_IDs[5],24,8) BTD(Common_Data.ReceiveData[153],0,Common_Data.Device_IDs[5],16,8) BTD(Common_Data.ReceiveData[154],0,Common_Data.Device_IDs[5],8,8) BTD(Common_Data.ReceiveData[155],0,Common_Data.Device_IDs[5],0,8) ,BTD(Common_Data.ReceiveData[178],0,Common_Data.Vendor_IDs[6],8,8) BTD(Common_Data.ReceiveData[179],0,Common_Data.Vendor_IDs[6],0,8) ,BTD(Common_Data.ReceiveData[180],0,Common_Data.Device_IDs[6],24,8) BTD(Common_Data.ReceiveData[181],0,Common_Data.Device_IDs[6],16,8) BTD(Common_Data.ReceiveData[182],0,Common_Data.Device_IDs[6],8,8) BTD(Common_Data.ReceiveData[183],0,Common_Data.Device_IDs[6],0,8) ,BTD(Common_Data.ReceiveData[206],0,Common_Data.Vendor_IDs[7],8,8) BTD(Common_Data.ReceiveData[207],0,Common_Data.Vendor_IDs[7],0,8) ,BTD(Common_Data.ReceiveData[208],0,Common_Data.Device_IDs[7],24,8) BTD(Common_Data.ReceiveData[209],0,Common_Data.Device_IDs[7],16,8) BTD(Common_Data.ReceiveData[210],0,Common_Data.Device_IDs[7],8,8) BTD(Common_Data.ReceiveData[211],0,Common_Data.Device_IDs[7],0,8) ,MOV(0,Status) ,MOV(TBEN_I_DATA[2],Prev_Input_Data_Valids) ];
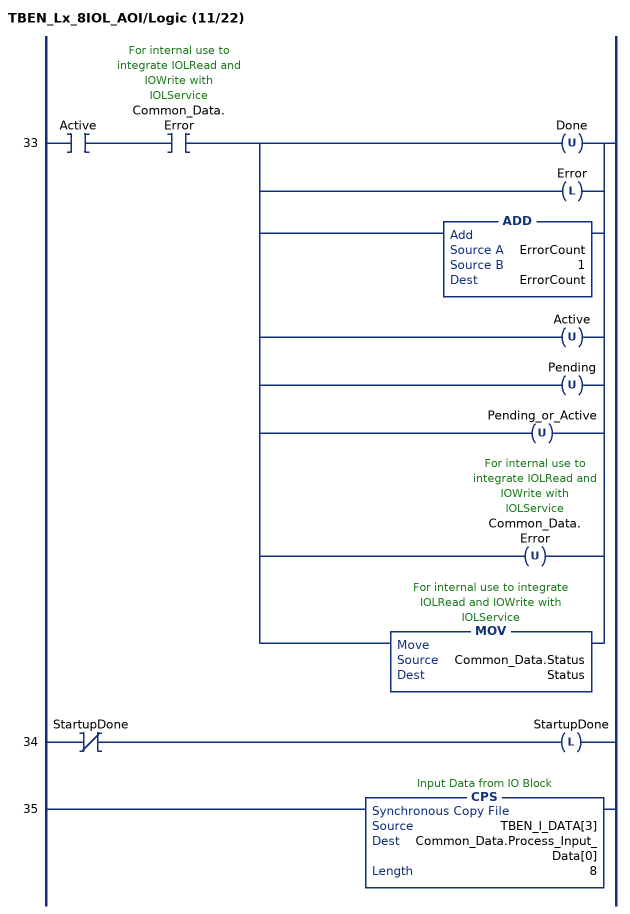
   33: XIC(Active)XIC(Common_Data.Error)[OTU(Done) ,OTL(Error) ,ADD(ErrorCount,1,ErrorCount) ,OTU(Active) ,OTU(Pending) ,OTU(Pending_or_Active) ,OTU(Common_Data.Error) ,MOV(Common_Data.Status,Status) ];
   34: XIO(StartupDone)OTL(StartupDone);
   35: CPS(TBEN_I_DATA[3],Common_Data.Process_Input_Data[0],8);
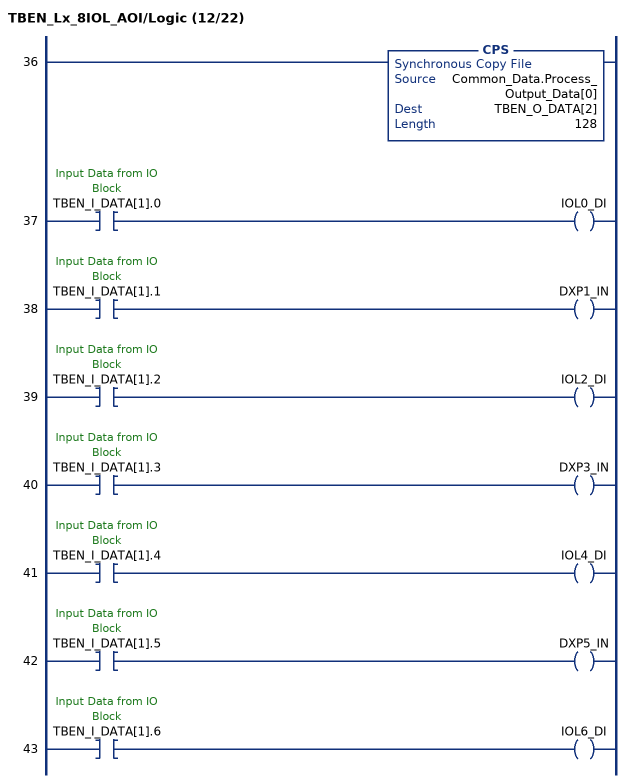
   36: CPS(Common_Data.Process_Output_Data[0],TBEN_O_DATA[2],128);
   37: XIC(TBEN_I_DATA[1].0)OTE(IOL0_DI);
   38: XIC(TBEN_I_DATA[1].1)OTE(DXP1_IN);
   39: XIC(TBEN_I_DATA[1].2)OTE(IOL2_DI);
   40: XIC(TBEN_I_DATA[1].3)OTE(DXP3_IN);
   41: XIC(TBEN_I_DATA[1].4)OTE(IOL4_DI);
   42: XIC(TBEN_I_DATA[1].5)OTE(DXP5_IN);
   43: XIC(TBEN_I_DATA[1].6)OTE(IOL6_DI);
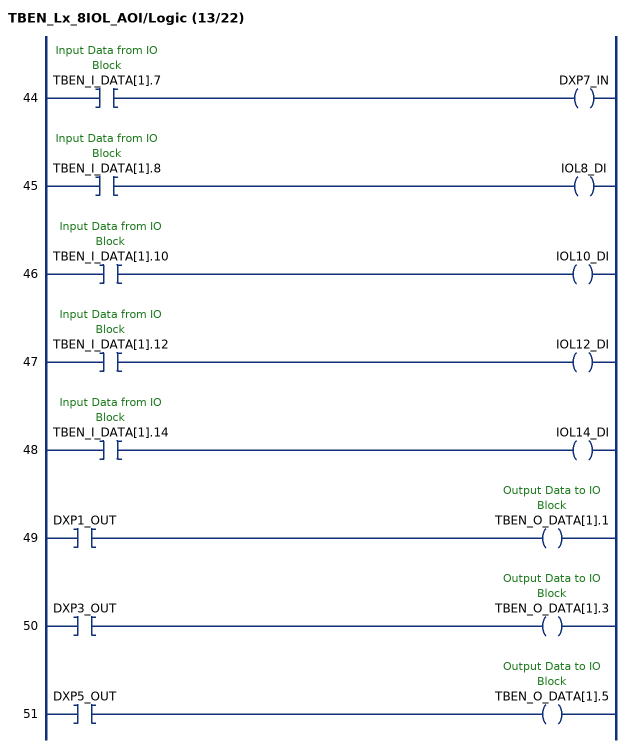
   44: XIC(TBEN_I_DATA[1].7)OTE(DXP7_IN);
   45: XIC(TBEN_I_DATA[1].8)OTE(IOL8_DI);
   46: XIC(TBEN_I_DATA[1].10)OTE(IOL10_DI);
   47: XIC(TBEN_I_DATA[1].12)OTE(IOL12_DI);
   48: XIC(TBEN_I_DATA[1].14)OTE(IOL14_DI);
   49: XIC(DXP1_OUT)OTE(TBEN_O_DATA[1].1);
   50: XIC(DXP3_OUT)OTE(TBEN_O_DATA[1].3);
   51: XIC(DXP5_OUT)OTE(TBEN_O_DATA[1].5);
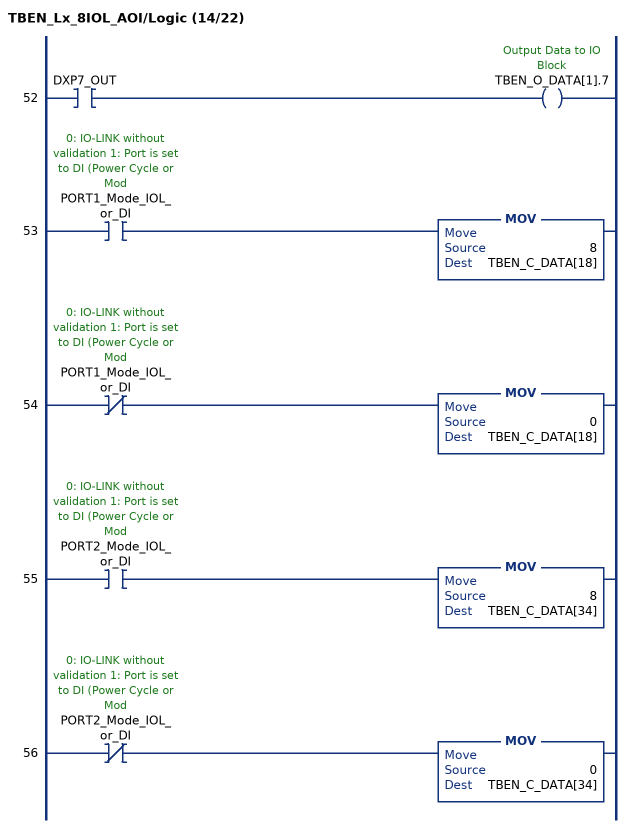
   52: XIC(DXP7_OUT)OTE(TBEN_O_DATA[1].7);
   53: XIC(PORT1_Mode_IOL_or_DI)MOV(8,TBEN_C_DATA[18]);
   54: XIO(PORT1_Mode_IOL_or_DI)MOV(0,TBEN_C_DATA[18]);
   55: XIC(PORT2_Mode_IOL_or_DI)MOV(8,TBEN_C_DATA[34]);
   56: XIO(PORT2_Mode_IOL_or_DI)MOV(0,TBEN_C_DATA[34]);
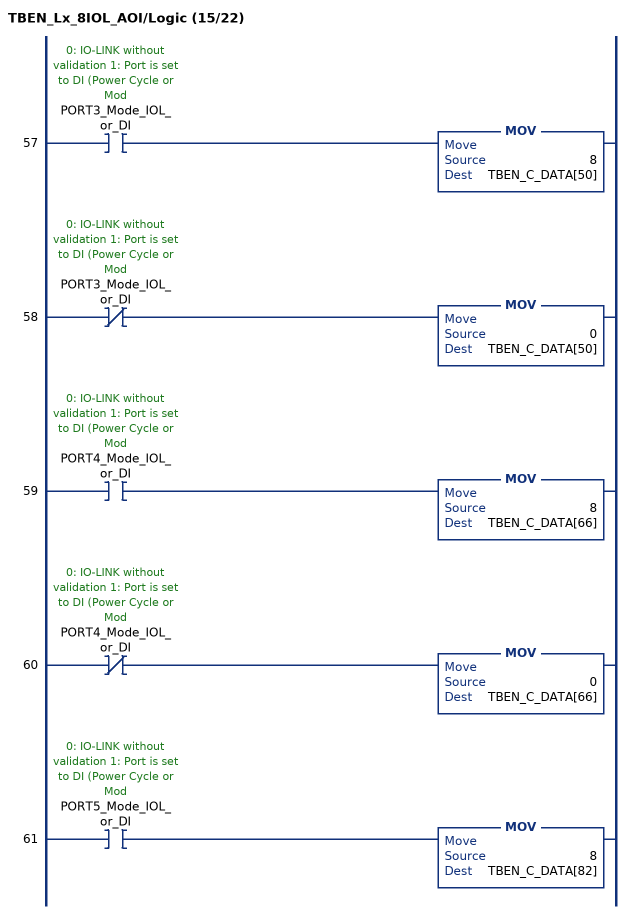
   57: XIC(PORT3_Mode_IOL_or_DI)MOV(8,TBEN_C_DATA[50]);
   58: XIO(PORT3_Mode_IOL_or_DI)MOV(0,TBEN_C_DATA[50]);
   59: XIC(PORT4_Mode_IOL_or_DI)MOV(8,TBEN_C_DATA[66]);
   60: XIO(PORT4_Mode_IOL_or_DI)MOV(0,TBEN_C_DATA[66]);
   61: XIC(PORT5_Mode_IOL_or_DI)MOV(8,TBEN_C_DATA[82]);
